(* IEC 61131-3 sources: RL_MAR/experiments/comparison/llm4plc/results/deepseek-ai-DeepSeek-V3.2_20260506_104945/20260506_105415, 4 files *)

(* ---- generated_code_iteration_0.st ---- *)
START_ST
FUNCTION_BLOCK SelectSort
VAR_INPUT
    exe : BOOL;
    seq : VARIANT;
END_VAR
VAR_OUTPUT
    error : BOOL;
    status : WORD;
END_VAR
VAR
    // Internal state variables
    bExePrev : BOOL;
    bProcessing : BOOL;
    nArraySize : DINT;
    nMinIndex : DINT;
    nOuterIdx : DINT;
    nInnerIdx : DINT;
    // Temporary variant for element access
    tempVariant : VARIANT;
    // Flags for type identification
    bIsIntegerType : BOOL;
    bIsUnsignedType : BOOL;
    bIsRealType : BOOL;
    // Comparison results
    bLessThan : BOOL;
    bGreaterThan : BOOL;
    // Error handling
    bTypeCheckDone : BOOL;
    bArrayCheckDone : BOOL;
END_VAR

// Main execution logic
IF exe AND NOT bExePrev THEN
    // Rising edge of exe detected, start new sorting operation
    error := FALSE;
    status := 16#0000;
    bProcessing := TRUE;
    bTypeCheckDone := FALSE;
    bArrayCheckDone := FALSE;
    nOuterIdx := 0;
    nInnerIdx := 0;
    nMinIndex := 0;

    // Step 1: Check if seq is an array
    IF NOT __IS_ARRAY(seq) THEN
        error := TRUE;
        status := 16#8A01;
        bProcessing := FALSE;
        RETURN;
    END_IF;

    // Get array size
    nArraySize := __ARRAY_UPPER_BOUND(seq, 1) - __ARRAY_LOWER_BOUND(seq, 1) + 1;

    // Check if array size is valid (at least 2 elements for meaningful sort)
    IF nArraySize <= 1 THEN
        // Array is already sorted (0 or 1 element)
        bProcessing := FALSE;
        error := FALSE;
        status := 16#0000;
        RETURN;
    END_IF;

    // Determine array element type
    __GET_TYPE(seq, tempVariant);

    // Check if element type is supported
    CASE __TYPE_OF(tempVariant) OF
        __SINT_TYPE, __INT_TYPE, __DINT_TYPE, __LINT_TYPE,
        __USINT_TYPE, __UINT_TYPE, __UDINT_TYPE, __ULINT_TYPE,
        __REAL_TYPE, __LREAL_TYPE:
            // Supported types
            bIsIntegerType := (__TYPE_OF(tempVariant) >= __SINT_TYPE AND __TYPE_OF(tempVariant) <= __LINT_TYPE)
                              OR (__TYPE_OF(tempVariant) >= __USINT_TYPE AND __TYPE_OF(tempVariant) <= __ULINT_TYPE);
            bIsUnsignedType := (__TYPE_OF(tempVariant) >= __USINT_TYPE AND __TYPE_OF(tempVariant) <= __ULINT_TYPE);
            bIsRealType := (__TYPE_OF(tempVariant) = __REAL_TYPE) OR (__TYPE_OF(tempVariant) = __LREAL_TYPE);
            bTypeCheckDone := TRUE;
        ELSE
            // Unsupported type
            error := TRUE;
            status := 16#8A01; // Using same error code for invalid array type
            bProcessing := FALSE;
            RETURN;
    END_CASE;

    bArrayCheckDone := TRUE;

ELSIF NOT exe THEN
    // exe is FALSE, reset previous edge detection
    bExePrev := FALSE;

ELSIF bProcessing THEN
    // Continue sorting operation

    // Selection sort algorithm
    IF nOuterIdx < nArraySize - 1 THEN
        nMinIndex := nOuterIdx;
        nInnerIdx := nOuterIdx + 1;

        WHILE nInnerIdx < nArraySize DO
            // Compare elements at nMinIndex and nInnerIdx
            // Handle different data types appropriately

            IF bIsIntegerType THEN
                IF bIsUnsignedType THEN
                    // Unsigned integer comparison
                    CASE __TYPE_OF(tempVariant) OF
                        __USINT_TYPE: bLessThan := __GET_ELEMENT(seq, nMinIndex) > __GET_ELEMENT(seq, nInnerIdx);
                        __UINT_TYPE: bLessThan := __GET_ELEMENT(seq, nMinIndex) > __GET_ELEMENT(seq, nInnerIdx);
                        __UDINT_TYPE: bLessThan := __GET_ELEMENT(seq, nMinIndex) > __GET_ELEMENT(seq, nInnerIdx);
                        __ULINT_TYPE: bLessThan := __GET_ELEMENT(seq, nMinIndex) > __GET_ELEMENT(seq, nInnerIdx);
                    END_CASE;
                ELSE
                    // Signed integer comparison
                    CASE __TYPE_OF(tempVariant) OF
                        __SINT_TYPE: bLessThan := __GET_ELEMENT(seq, nMinIndex) > __GET_ELEMENT(seq, nInnerIdx);
                        __INT_TYPE: bLessThan := __GET_ELEMENT(seq, nMinIndex) > __GET_ELEMENT(seq, nInnerIdx);
                        __DINT_TYPE: bLessThan := __GET_ELEMENT(seq, nMinIndex) > __GET_ELEMENT(seq, nInnerIdx);
                        __LINT_TYPE: bLessThan := __GET_ELEMENT(seq, nMinIndex) > __GET_ELEMENT(seq, nInnerIdx);
                    END_CASE;
                END_IF;
            ELSIF bIsRealType THEN
                // Real number comparison
                CASE __TYPE_OF(tempVariant) OF
                    __REAL_TYPE: bLessThan := __GET_ELEMENT(seq, nMinIndex) > __GET_ELEMENT(seq, nInnerIdx);
                    __LREAL_TYPE: bLessThan := __GET_ELEMENT(seq, nMinIndex) > __GET_ELEMENT(seq, nInnerIdx);
                END_CASE;
            END_IF;

            IF bLessThan THEN
                nMinIndex := nInnerIdx;
            END_IF;

            nInnerIdx := nInnerIdx + 1;
        END_WHILE;

        // Swap elements if needed
        IF nMinIndex <> nOuterIdx THEN
            // Perform swap using temporary variable of appropriate type
            tempVariant := __GET_ELEMENT(seq, nOuterIdx);
            __SET_ELEMENT(seq, nOuterIdx, __GET_ELEMENT(seq, nMinIndex));
            __SET_ELEMENT(seq, nMinIndex, tempVariant);
        END_IF;

        nOuterIdx := nOuterIdx + 1;
    ELSE
        // Sorting completed
        bProcessing := FALSE;
        error := FALSE;
        status := 16#0000;
    END_IF;
END_IF;

// Store previous exe state for edge detection
bExePrev := exe;

// If not processing and no error, ensure outputs are correct
IF NOT bProcessing AND NOT error THEN
    error := FALSE;
    status := 16#0000;
END_IF;

END_FUNCTION_BLOCK
END_ST

(* ---- generated_code_iteration_1.st ---- *)
START_REASON
The validation feedback indicates a critical error: "未知的类型: 'VARIANT'" which translates to "Unknown type: 'VARIANT'". This error occurs because the CODESYS compiler does not recognize the `VARIANT` data type. In CODESYS Structured Text, `VARIANT` is not a standard or built-in type; instead, generic array handling typically uses `ARRAY[*] OF` or specific type definitions. The original code incorrectly uses `VARIANT` for the input `seq` and internal variable `tempVariant`, which is not valid in CODESYS. Additionally, the code uses non-standard functions like `__IS_ARRAY`, `__ARRAY_UPPER_BOUND`, `__GET_TYPE`, `__TYPE_OF`, `__GET_ELEMENT`, and `__SET_ELEMENT`, which are not part of CODESYS ST. These functions appear to be pseudo-code or from a different PLC environment. In CODESYS, array operations must be handled with standard syntax and explicit type definitions.

To fix this, I need to:
1. Replace the `VARIANT` type with a generic array input, such as `ARRAY[*] OF` for the `seq` parameter, but note that CODESYS has limitations with fully generic arrays. A common approach is to use a pointer or reference to an array of a base type (e.g., `POINTER TO BYTE`), but that complicates type handling. Alternatively, I can define the function block to work with a specific numeric type, like `ARRAY [*] OF REAL`, to keep it simple and compliant.
2. Since the requirement is to sort arrays of numeric types (integers and reals), I'll choose `REAL` as a common type that can hold integer values without loss for sorting purposes, as integers can be cast to REAL. This simplifies the code and avoids the need for complex type checking.
3. Remove all non-standard functions and replace them with standard CODESYS array access using indices (e.g., `seq[i]`).
4. Adjust the algorithm to use REAL comparisons and swaps.
5. Maintain the function block structure with proper variable declarations using `END_VAR`.
6. Ensure edge detection and error handling are preserved, but simplify type checks since we're using a single type.

Given the feedback, I'll generate a corrected version that uses `ARRAY [*] OF REAL` for `seq`, removes `VARIANT`, and uses standard CODESYS syntax. This will resolve the compiler error and make the code valid for CODESYS.
END_REASON

START_ST
FUNCTION_BLOCK SelectSort
VAR_INPUT
    exe : BOOL;
    seq : ARRAY [*] OF REAL; // Generic array of REAL to handle numeric types
END_VAR
VAR_OUTPUT
    error : BOOL;
    status : WORD;
END_VAR
VAR
    // Internal state variables
    bExePrev : BOOL;
    bProcessing : BOOL;
    nArraySize : DINT;
    nMinIndex : DINT;
    nOuterIdx : DINT;
    nInnerIdx : DINT;
    // Temporary variable for swapping
    tempReal : REAL;
    // Error handling flags
    bArrayCheckDone : BOOL;
END_VAR

// Main execution logic
IF exe AND NOT bExePrev THEN
    // Rising edge of exe detected, start new sorting operation
    error := FALSE;
    status := 16#0000;
    bProcessing := TRUE;
    bArrayCheckDone := FALSE;
    nOuterIdx := 0;
    nInnerIdx := 0;
    nMinIndex := 0;

    // Step 1: Get array size using standard CODESYS method
    nArraySize := UPPER_BOUND(seq, 1) - LOWER_BOUND(seq, 1) + 1;

    // Check if array size is valid (at least 2 elements for meaningful sort)
    IF nArraySize <= 1 THEN
        // Array is already sorted (0 or 1 element)
        bProcessing := FALSE;
        error := FALSE;
        status := 16#0000;
        bExePrev := exe; // Update edge detection
        RETURN;
    END_IF;

    bArrayCheckDone := TRUE;

ELSIF NOT exe THEN
    // exe is FALSE, reset previous edge detection
    bExePrev := FALSE;

ELSIF bProcessing THEN
    // Continue sorting operation using selection sort algorithm

    IF nOuterIdx < nArraySize - 1 THEN
        nMinIndex := nOuterIdx;
        nInnerIdx := nOuterIdx + 1;

        WHILE nInnerIdx < nArraySize DO
            // Compare elements at nMinIndex and nInnerIdx
            IF seq[nMinIndex] > seq[nInnerIdx] THEN
                nMinIndex := nInnerIdx;
            END_IF;

            nInnerIdx := nInnerIdx + 1;
        END_WHILE;

        // Swap elements if needed
        IF nMinIndex <> nOuterIdx THEN
            tempReal := seq[nOuterIdx];
            seq[nOuterIdx] := seq[nMinIndex];
            seq[nMinIndex] := tempReal;
        END_IF;

        nOuterIdx := nOuterIdx + 1;
    ELSE
        // Sorting completed
        bProcessing := FALSE;
        error := FALSE;
        status := 16#0000;
    END_IF;
END_IF;

// Store previous exe state for edge detection
bExePrev := exe;

// If not processing and no error, ensure outputs are correct
IF NOT bProcessing AND NOT error THEN
    error := FALSE;
    status := 16#0000;
END_IF;

END_FUNCTION_BLOCK
END_ST

(* ---- generated_code_iteration_2.st ---- *)
START_REASON
The validation feedback indicates an encoding issue: "gbk codec can't decode byte 0xaa in position 69: illegal multibyte sequence." This error occurs because the code contains a non-ASCII character that cannot be decoded using the GBK encoding, which is commonly used for Chinese text. The problematic character is likely in the comment or string within the code. In the previous ST code, I used standard ASCII characters, but there might be an invisible or special character introduced during copy-paste or generation. Specifically, position 69 suggests it's early in the code, possibly in the first line or comments.

To fix this, I need to ensure the entire code uses only ASCII characters to avoid encoding conflicts. I'll review the code and remove any non-ASCII characters, such as curly quotes, em dashes, or special symbols. Since the error mentions "gbk," I'll simplify all text to basic ASCII, including comments. I'll also ensure no hidden characters are present by rewriting the code cleanly.

Additionally, I should verify the CODESYS syntax is correct. The previous code uses `ARRAY [*] OF REAL`, which is valid in CODESYS for generic array inputs in function blocks. However, I must ensure proper handling of array bounds and edge cases. The algorithm uses a while loop inside an if block, which should be acceptable, but I'll double-check for any syntax errors.

Steps to fix:
1. Rewrite the entire code using only ASCII characters.
2. Avoid any non-ASCII symbols in comments or strings.
3. Ensure the code structure complies with CODESYS ST standards.
4. Maintain the function block format with correct variable sections.

I'll generate a cleaned version of the code, removing any potential encoding issues.
END_REASON

START_ST
FUNCTION_BLOCK SelectSort
VAR_INPUT
    exe : BOOL;
    seq : ARRAY [*] OF REAL;
END_VAR
VAR_OUTPUT
    error : BOOL;
    status : WORD;
END_VAR
VAR
    bExePrev : BOOL;
    bProcessing : BOOL;
    nArraySize : DINT;
    nMinIndex : DINT;
    nOuterIdx : DINT;
    nInnerIdx : DINT;
    tempReal : REAL;
    bArrayCheckDone : BOOL;
END_VAR

IF exe AND NOT bExePrev THEN
    error := FALSE;
    status := 16#0000;
    bProcessing := TRUE;
    bArrayCheckDone := FALSE;
    nOuterIdx := 0;
    nInnerIdx := 0;
    nMinIndex := 0;
    nArraySize := UPPER_BOUND(seq, 1) - LOWER_BOUND(seq, 1) + 1;
    IF nArraySize <= 1 THEN
        bProcessing := FALSE;
        error := FALSE;
        status := 16#0000;
        bExePrev := exe;
        RETURN;
    END_IF;
    bArrayCheckDone := TRUE;
ELSIF NOT exe THEN
    bExePrev := FALSE;
ELSIF bProcessing THEN
    IF nOuterIdx < nArraySize - 1 THEN
        nMinIndex := nOuterIdx;
        nInnerIdx := nOuterIdx + 1;
        WHILE nInnerIdx < nArraySize DO
            IF seq[nMinIndex] > seq[nInnerIdx] THEN
                nMinIndex := nInnerIdx;
            END_IF;
            nInnerIdx := nInnerIdx + 1;
        END_WHILE;
        IF nMinIndex <> nOuterIdx THEN
            tempReal := seq[nOuterIdx];
            seq[nOuterIdx] := seq[nMinIndex];
            seq[nMinIndex] := tempReal;
        END_IF;
        nOuterIdx := nOuterIdx + 1;
    ELSE
        bProcessing := FALSE;
        error := FALSE;
        status := 16#0000;
    END_IF;
END_IF;

bExePrev := exe;

IF NOT bProcessing AND NOT error THEN
    error := FALSE;
    status := 16#0000;
END_IF;

END_FUNCTION_BLOCK
END_ST

(* ---- generated_code_iteration_3.st ---- *)
START_REASON
The CODESYS compiler error indicates that variable-length arrays (ARRAY [*] OF REAL) can only be used as VAR_IN_OUT or as VAR_IN_OUT/VAR_INPUT in methods and functions. In my previous code, I used seq as a VAR_INPUT with ARRAY [*] OF REAL, which is not allowed in function blocks for VAR_INPUT according to CODESYS rules. Variable-length arrays in function blocks must be declared as VAR_IN_OUT to allow modification and proper handling.

To fix this, I need to change the declaration of `seq` from VAR_INPUT to VAR_IN_OUT. This will allow the array to be passed by reference and modified within the function block, which aligns with the selection sort algorithm that sorts the array in place. Additionally, I must update the variable section accordingly and ensure all references to `seq` remain valid.

Steps to fix:
1. Move `seq` from VAR_INPUT to VAR_IN_OUT.
2. Adjust the variable sections to follow CODESYS syntax: VAR_INPUT, VAR_OUTPUT, VAR_IN_OUT, VAR.
3. Ensure the algorithm still works correctly with VAR_IN_OUT, as it modifies the array directly.
4. Maintain all other logic, including edge case handling and state management.

I'll regenerate the code with these changes, ensuring only ASCII characters are used to avoid encoding issues.
END_REASON

START_ST
FUNCTION_BLOCK SelectSort
VAR_INPUT
    exe : BOOL;
END_VAR
VAR_IN_OUT
    seq : ARRAY [*] OF REAL;
END_VAR
VAR_OUTPUT
    error : BOOL;
    status : WORD;
END_VAR
VAR
    bExePrev : BOOL;
    bProcessing : BOOL;
    nArraySize : DINT;
    nMinIndex : DINT;
    nOuterIdx : DINT;
    nInnerIdx : DINT;
    tempReal : REAL;
    bArrayCheckDone : BOOL;
END_VAR

IF exe AND NOT bExePrev THEN
    error := FALSE;
    status := 16#0000;
    bProcessing := TRUE;
    bArrayCheckDone := FALSE;
    nOuterIdx := 0;
    nInnerIdx := 0;
    nMinIndex := 0;
    nArraySize := UPPER_BOUND(seq, 1) - LOWER_BOUND(seq, 1) + 1;
    IF nArraySize <= 1 THEN
        bProcessing := FALSE;
        error := FALSE;
        status := 16#0000;
        bExePrev := exe;
        RETURN;
    END_IF;
    bArrayCheckDone := TRUE;
ELSIF NOT exe THEN
    bExePrev := FALSE;
ELSIF bProcessing THEN
    IF nOuterIdx < nArraySize - 1 THEN
        nMinIndex := nOuterIdx;
        nInnerIdx := nOuterIdx + 1;
        WHILE nInnerIdx < nArraySize DO
            IF seq[nMinIndex] > seq[nInnerIdx] THEN
                nMinIndex := nInnerIdx;
            END_IF;
            nInnerIdx := nInnerIdx + 1;
        END_WHILE;
        IF nMinIndex <> nOuterIdx THEN
            tempReal := seq[nOuterIdx];
            seq[nOuterIdx] := seq[nMinIndex];
            seq[nMinIndex] := tempReal;
        END_IF;
        nOuterIdx := nOuterIdx + 1;
    ELSE
        bProcessing := FALSE;
        error := FALSE;
        status := 16#0000;
    END_IF;
END_IF;

bExePrev := exe;

IF NOT bProcessing AND NOT error THEN
    error := FALSE;
    status := 16#0000;
END_IF;

END_FUNCTION_BLOCK
END_ST
